FUNCTION_BLOCK AX_INTERLOCK_2 (* Event-driven bistable and Toggle with Dual Interlock *)
  (* Standard: 61499-1 Annex A; Description: Copyright (c) 2017, 2024 fortiss GmbH, HR Agrartechnik GmbH This program and the accompanying materials are made available under the terms of the Eclipse Public License 2.0 which is available at https://www.eclipse.org/legal/epl-2.0/ SPDX-License-Identifier: EPL-2.0 *)
  (* Version 3.0, 2025-04-14, Patrick Aigner, changed package *)
  (* Version 1.1, 2024-08-27, Franz Höpfinger, HR Agrartechnik GmbH, Copy E_SR and make this FB *)
  (* Version 1.0, 2017-09-22, Alois Zoitl, fortiss GmbH, initial API and implementation and/or initial documentation *)
  PACKAGE logiBUS::utils::interlock;
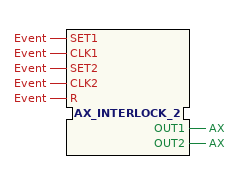
  EVENT_INPUT
    SET1; (* Set output OUT1 *)
    CLK1; (* Clock for triggering a output toggle on OUT1 *)
    SET2; (* Set output OUT2 *)
    CLK2; (* Clock for triggering a output toggle on OUT2 *)
    R; (* Reset all outputs *)
  END_EVENT
  PLUGS
    OUT1 : adapter::types::unidirectional::AX; (* value of flip flop *)
    OUT2 : adapter::types::unidirectional::AX; (* value of flip flop *)
  END_PLUGS
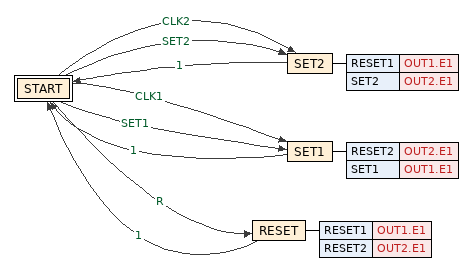
  EC_STATES
    START; (* Initial State *)
    SET1 : RESET2 -> OUT2.E1, SET1 -> OUT1.E1;
    RESET : RESET1 -> OUT1.E1, RESET2 -> OUT2.E1;
    SET2 : RESET1 -> OUT1.E1, SET2 -> OUT2.E1;
  END_STATES
  EC_TRANSITIONS
    START TO SET1 := SET1;
    START TO SET2 := SET2;
    START TO SET1 := CLK1;
    START TO SET2 := CLK2;
    START TO RESET := R;
    SET1 TO START := 1;
    SET2 TO START := 1;
    RESET TO START := 1;
  END_TRANSITIONS
  ALGORITHM SET1 IN ST:
OUT1.D1 := TRUE;
  END_ALGORITHM
  ALGORITHM SET2 IN ST:
OUT2.D1 := TRUE;
  END_ALGORITHM
  ALGORITHM RESET1 IN ST:
OUT1.D1 := FALSE;
  END_ALGORITHM
  ALGORITHM RESET2 IN ST:
OUT2.D1 := FALSE;
  END_ALGORITHM
END_FUNCTION_BLOCK
